{attribute addProperty BoxType "EL3255-0000-0016"}
{attribute addProperty Id "RTD_Standard_ChannelAT %I*ARRAY[0..8] OF RTD_Standard_Channel_904746A2160200WcStateAT %I*WcState_98A4DF7520.250InfoDataAT %I*InfoData_BC63D37F80100"}
{attribute addProperty CRC "3458581715"}
{attribute addProperty SizeInBites "242"}
{attribute addProperty SizeInBytes "30.25"}
TYPE EL3255_6616AD46 :
STRUCT
	{attribute addProperty Name "RTD_Standard_Channel"}
	RTD_Standard_Channel : ARRAY[0..8] OF RTD_Standard_Channel_904746A2;
	{attribute addProperty Name "WcState"}
	WcState : WcState_98A4DF75;
	{attribute addProperty Name "InfoData"}
	InfoData : InfoData_BC63D37F;
END_STRUCT
END_TYPE

(* stored: Version 1.2.0.0, ProductVersion 3.1.4024.9
   DUT EL3255_6616AD46: Id {0c7d3feb-57a4-4cda-9384-72f12403e9b6} *)
